TYPE ST_GearAxis_1 :
STRUCT
    nIndex: UINT := 1; //Index of the master axis
    fRatio: LREAL := 0; //Gearing ratio between master axis and this one
END_STRUCT
END_TYPE

(* stored: Version 1.1.0.1, ProductVersion 3.1.4024.6
   DUT ST_GearAxis_1: Id {4039494b-a915-420d-a0fe-2a0ffe7180a9} *)
